(* PLC project SafeLOGIC-1, BrAutomation SafeDESIGNER  4.3.2.11 *)
(* stored: companyURL http://www.br-automation.com, creationDateTime Wed Jun 13 14:03:58 2018 *)

PROGRAM Main

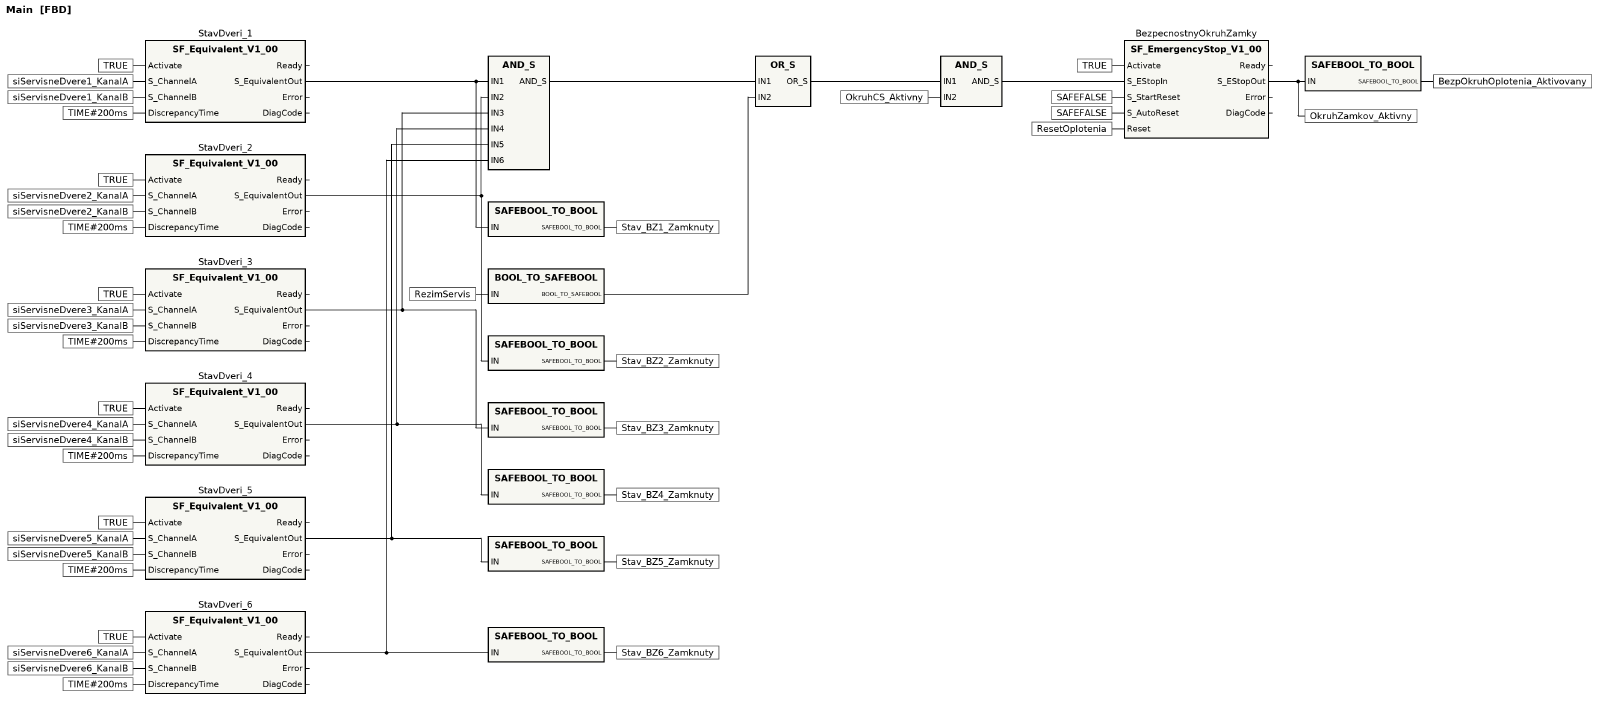
(* FBD diagram, written out as Structured Text *)
StavDveri_1(Activate := TRUE, S_ChannelA := siServisneDvere1_KanalA, S_ChannelB := siServisneDvere1_KanalB, DiscrepancyTime := TIME#200ms);
Stav_BZ1_Zamknuty := SAFEBOOL_TO_BOOL(StavDveri_1.S_EquivalentOut);
StavDveri_2(Activate := TRUE, S_ChannelA := siServisneDvere2_KanalA, S_ChannelB := siServisneDvere2_KanalB, DiscrepancyTime := TIME#200ms);
StavDveri_3(Activate := TRUE, S_ChannelA := siServisneDvere3_KanalA, S_ChannelB := siServisneDvere3_KanalB, DiscrepancyTime := TIME#200ms);
StavDveri_4(Activate := TRUE, S_ChannelA := siServisneDvere4_KanalA, S_ChannelB := siServisneDvere4_KanalB, DiscrepancyTime := TIME#200ms);
StavDveri_5(Activate := TRUE, S_ChannelA := siServisneDvere5_KanalA, S_ChannelB := siServisneDvere5_KanalB, DiscrepancyTime := TIME#200ms);
StavDveri_6(Activate := TRUE, S_ChannelA := siServisneDvere6_KanalA, S_ChannelB := siServisneDvere6_KanalB, DiscrepancyTime := TIME#200ms);
BezpecnostnyOkruhZamky(Activate := TRUE, S_EStopIn := AND_S(OR_S(AND_S(StavDveri_1.S_EquivalentOut, StavDveri_2.S_EquivalentOut, StavDveri_3.S_EquivalentOut, StavDveri_4.S_EquivalentOut, StavDveri_5.S_EquivalentOut, StavDveri_6.S_EquivalentOut), BOOL_TO_SAFEBOOL(RezimServis)), OkruhCS_Aktivny), S_StartReset := SAFEFALSE, S_AutoReset := SAFEFALSE, Reset := ResetOplotenia);
OkruhZamkov_Aktivny := BezpecnostnyOkruhZamky.S_EStopOut;
BezpOkruhOplotenia_Aktivovany := SAFEBOOL_TO_BOOL(BezpecnostnyOkruhZamky.S_EStopOut);
Stav_BZ2_Zamknuty := SAFEBOOL_TO_BOOL(StavDveri_2.S_EquivalentOut);
Stav_BZ3_Zamknuty := SAFEBOOL_TO_BOOL(StavDveri_3.S_EquivalentOut);
Stav_BZ4_Zamknuty := SAFEBOOL_TO_BOOL(StavDveri_4.S_EquivalentOut);
Stav_BZ5_Zamknuty := SAFEBOOL_TO_BOOL(StavDveri_5.S_EquivalentOut);
Stav_BZ6_Zamknuty := SAFEBOOL_TO_BOOL(StavDveri_6.S_EquivalentOut);
END_PROGRAM
